FUNCTION_BLOCK CallbackFB (* Composite FB for easy use of the Callback in Subapplications *)
  (* Standard: 61499-2 *)
  (* Version 1.0, 2025-09-06, Franz Höpfinger, initial API and implementation and/or initial documentation *)
  PACKAGE isobus::pgn::tx;
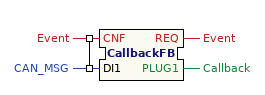
  EVENT_INPUT
    CNF WITH DI1; (* Confirmation from Plug *)
  END_EVENT
  EVENT_OUTPUT
    REQ; (* Request from Socket *)
  END_EVENT
  VAR_INPUT
    DI1 : isobus::pgn::CAN_MSG;
  END_VAR
  PLUGS
    PLUG1 : isobus::pgn::tx::Callback;
  END_PLUGS
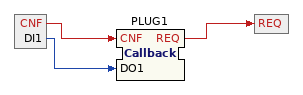
  EVENT_CONNECTIONS
    CNF TO PLUG1.CNF;
    PLUG1.REQ TO REQ;
  END_CONNECTIONS
  DATA_CONNECTIONS
    DI1 TO PLUG1.DO1;
  END_CONNECTIONS
END_FUNCTION_BLOCK
